(*
    This function compares two instances of any object type and returns whether they
    are the same type, size and value or not. This is necessary for two reasons:
    1. So that we can know exactly what differs between the two input parameters
    2. It's not possible to do a comparison (= or <>) between two instances of ANY.
*)
FUNCTION F_AnyComparator
VAR_INPUT
    AnyValueOne : ANY;
    AnyValueTwo : ANY;
END_VAR
VAR_OUTPUT
    bDataTypesNotEquals : BOOL; // The data type of the two ANY input parameters are not equal
    bDataSizeNotEquals : BOOL; // The data size of the two ANY input parameters are not equal
    bDataContentNotEquals : BOOL; // The data content of the two ANY input parameters are not equal
END_VAR
VAR
    nCount : DINT;
END_VAR

(* Check whether the type of the inputs differs *)
IF AnyValueOne.TypeClass <> AnyValueTwo.TypeClass THEN
    bDataTypesNotEquals := TRUE;
END_IF

(* Check whether the size of the inputs differs *)
IF NOT bDataTypesNotEquals THEN
    IF (AnyValueOne.diSize <> AnyValueTwo.diSize) THEN
        bDataSizeNotEquals := TRUE;
    END_IF
END_IF

(* Even though the data type and size are equals, the contents may still differ *)
IF NOT bDataTypesNotEquals AND NOT bDataSizeNotEquals THEN
    (* Compare each byte in the ANY-types *)
    FOR nCount := 0 TO AnyValueOne.diSize-1 BY 1 DO
        IF (UDINT_TO_DINT(AnyValueOne.TypeClass) = IBaseLibrary.TYPE_STRING) OR
            (UDINT_TO_DINT(AnyValueOne.TypeClass) = IBaseLibrary.TYPE_WSTRING) THEN
            IF F_ToChr(c := AnyValueOne.pValue[nCount]) = '$00' THEN
                EXIT;
            END_IF
        END_IF

        IF AnyValueOne.pValue[nCount] <> AnyValueTwo.pValue[nCount] THEN
            bDataContentNotEquals := TRUE;
            EXIT;
        END_IF
    END_FOR
END_IF

END_FUNCTION

(* stored: Version 1.1.0.1, ProductVersion 3.1.4022.12
   POU F_AnyComparator: Id {e4f95c0d-0ece-47a8-977f-f9d45a4f920e}, SpecialFunc None *)
